// Mitsubishi GX Works2 project: test   PLC: FX3U/FX3UC

PROGRAM MAIN
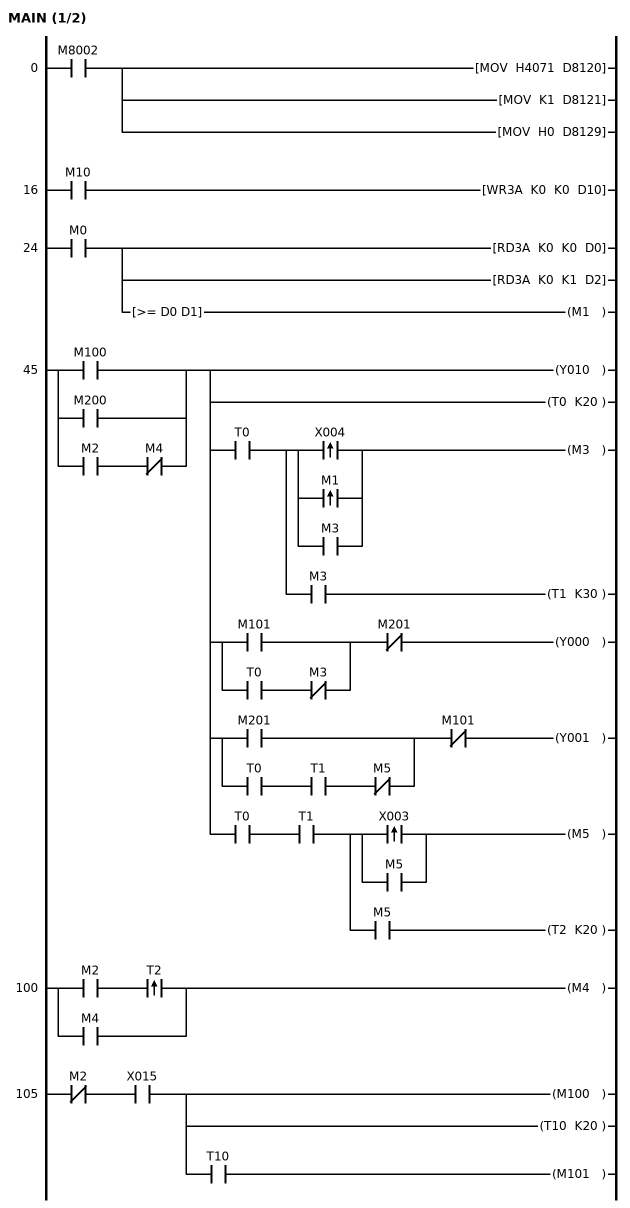
0     LD      M8002
      MOV     H4071 D8120
      MOV     K1 D8121
      MOV     H0 D8129
16    LD      M10
      WR3A    K0 K0 D10
24    LD      M0
      RD3A    K0 K0 D0
      RD3A    K0 K1 D2
      AND>=   D0 D1
      OUT     M1
45    LD      M100
      OR      M200
      LD      M2
      ANI     M4
      ORB
      OUT     Y010
      OUT     T0 K20
      MPS
      AND     T0
      MPS
      LDP     X004
      ORP     M1
      OR      M3
      ANB
      OUT     M3
      MPP
      AND     M3
      OUT     T1 K30
      MRD
      LD      M101
      LD      T0
      ANI     M3
      ORB
      ANB
      ANI     M201
      OUT     Y000
      MRD
      LD      M201
      LD      T0
      AND     T1
      ANI     M5
      ORB
      ANB
      ANI     M101
      OUT     Y001
      MPP
      AND     T0
      AND     T1
      MPS
      LDP     X003
      OR      M5
      ANB
      OUT     M5
      MPP
      AND     M5
      OUT     T2 K20
100   LD      M2
      ANDP    T2
      OR      M4
      OUT     M4
105   LDI     M2
      AND     X015
      OUT     M100
      OUT     T10 K20
      AND     T10
      OUT     M101
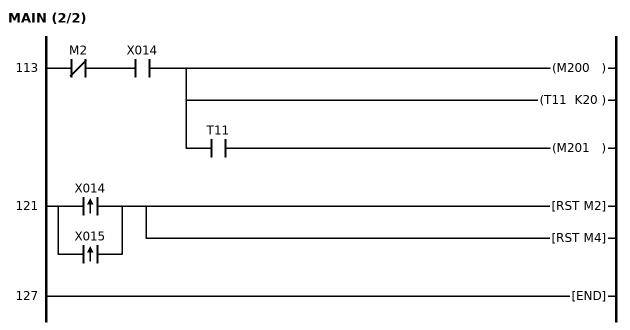
113   LDI     M2
      AND     X014
      OUT     M200
      OUT     T11 K20
      AND     T11
      OUT     M201
121   LDP     X014
      ORP     X015
      RST     M2
      RST     M4
127   END
END_PROGRAM
